SUBAPPLICATION Button_IXA_TO_logiBUS_QXA_BG_OPC (* Button IXA -> logiBUS QXA + Hintergrundfarbe, plus OPC-UA Read/Write (generisch, ein Kanal) *)
  (* Standard: 61499-2; Description: Copyright (c) 2023 Meisterschulen am Ostbahnhof This program and the accompanying materials are made available under the terms of the Eclipse Public License 2.0 which is available at https://www.eclipse.org/legal/epl-2.0/ SPDX-License-Identifier: EPL-2.0 *)
  (* Version 1.2, 2026-09-07, Franz Höpfinger, Meisterschulen am Ostbahnhof, Vorruebergehend non-latching: SR-Latch (AX_ASR_RF_TRIG x2 + ASR_MERGE_2 + ASR_AX_SR) durch einfaches AX_OR_2 ersetzt - Button UND Remote-Kommando sind jetzt tastend (Pegel), kein Klick-Toggle mehr *)
  (* Version 1.1, 2026-07-20, Franz Höpfinger, Meisterschulen am Ostbahnhof, Background *)
  (* Version 1.0, 2026-01-15, Franz Höpfinger, Meisterschulen am Ostbahnhof, initial API and implementation and/or initial documentation *)
  PACKAGE MyLib::sys;
  IMPORT isobus::UT::Q::const::IDs::ID_NULL;
  IMPORT logiBUS::io::DQ::logiBUS_DO;
  IMPORT logiBUS::io::DQ::logiBUS_DO_S;
  (* Documentation:
  Button → logiBUS-Ausgang, tastend (Pegel-ODER)
   Lokaler VT-Button UND Remote-OPC-UA-Kommando sind beides kontinuierliche Pegel (keine Events) - AX_OR_2 verknüpft sie direkt: der Ausgang ist EIN, solange irgendeine der beiden Quellen gerade aktiv ist, und fällt sofort wieder ab, sobald beide inaktiv sind. Kein Klick-Toggle, kein Latch, kein Stuck-On-Zustand.
   Für die vorherige Klick-Toggle-Variante (SR-Latch, ein Klick EIN, nächster Klick AUS) Button_IXA_TO_logiBUS_QXA_BG_OPC_LATCHING verwenden - identisches Interface, 1:1 austauschbar.
  *)
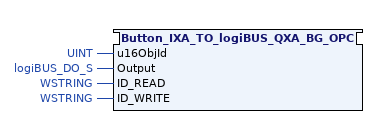
  VAR_INPUT
    u16ObjId : UINT := ID_NULL; (* Object ID Button/Hintergrund (VT), ID_NULL = noch kein VT-Objekt *)
    Output : logiBUS::io::DQ::logiBUS_DO_S := logiBUS_DO::Invalid; (* Identify the Output Output_Q1..Q12 *)
    ID_READ : WSTRING; (* OPC-UA Subscribe-Key (schreibbar) *)
    ID_WRITE : WSTRING; (* OPC-UA Publish-Key (lesbar) *)
  END_VAR
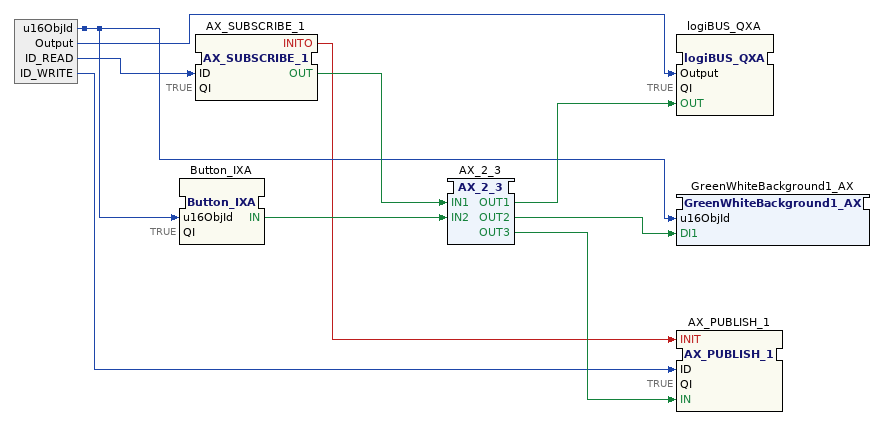
  FBS
    logiBUS_QXA : logiBUS::io::DQ::logiBUS_QXA(QI := TRUE);
    Button_IXA : isobus::UT::io::Button::Button_IXA(QI := TRUE);
    AX_SUBSCRIBE_1 : adapter::net::AX_SUBSCRIBE_1(QI := TRUE);
    AX_PUBLISH_1 : adapter::net::AX_PUBLISH_1(QI := TRUE);
  END_FBS
  SUBAPPS
    GreenWhiteBackground1_AX : MyLib::sys::GreenWhiteBackground1_AX;
    AX_2_3 : AX_2_3;
  END_SUBAPPS
  EVENT_CONNECTIONS
    AX_SUBSCRIBE_1.INITO TO AX_PUBLISH_1.INIT;
  END_CONNECTIONS
  DATA_CONNECTIONS
    u16ObjId TO Button_IXA.u16ObjId;
    Output TO logiBUS_QXA.Output;
    u16ObjId TO GreenWhiteBackground1_AX.u16ObjId;
    ID_READ TO AX_SUBSCRIBE_1.ID;
    ID_WRITE TO AX_PUBLISH_1.ID;
  END_CONNECTIONS
  ADAPTER_CONNECTIONS
    Button_IXA.IN TO AX_2_3.IN2;
    AX_SUBSCRIBE_1.OUT TO AX_2_3.IN1;
    AX_2_3.OUT1 TO logiBUS_QXA.OUT;
    AX_2_3.OUT2 TO GreenWhiteBackground1_AX.DI1;
    AX_2_3.OUT3 TO AX_PUBLISH_1.IN;
  END_CONNECTIONS
END_SUBAPPLICATION
